{attribute addProperty BoxType "KL6904-0001"}
{attribute addProperty Id "Channel_1Channel_43EA163900"}
{attribute addProperty CRC "105552965"}
{attribute addProperty SizeInBites "0"}
{attribute addProperty SizeInBytes "0"}
TYPE KL_064A9C45 :
STRUCT
	{attribute addProperty Name "Channel_1"}
	Channel_1 : Channel_43EA1639;
END_STRUCT
END_TYPE

(* stored: Version 1.2.0.0, ProductVersion 3.1.4024.9
   DUT KL_064A9C45: Id {17835288-e179-4c4a-a931-e00b7063d9d9} *)
